FUNCTION_BLOCK Robot_MH

VAR_INPUT
	Robot_1_In			: MH_Robot;
	Part_Unload_Comp	: BOOL;
END_VAR

VAR_OUTPUT
	Robot_1_Out			: MH_Robot;	
END_VAR

VAR
	Pickup_Delay			: ARRAY [0..5] OF TON;
END_VAR

CASE Robot_1_In.i_Prg_No OF
	101:
		IF (Robot_1_In.i_Home AND Robot_1_In.i_Area_Ok1 AND Robot_1_In.i_Start) THEN
		Pickup_Delay[0](IN:= Robot_1_In.i_Start, PT:= T#1S, Q=> , ET=> );
		IF Pickup_Delay[0].Q THEN
		Robot_1_In.i_Home := FALSE;
		Robot_1_Out.o_Pickup_Comp1 := TRUE;
		Robot_1_In.i_Home := TRUE;
		END_IF
		END_IF
		IF (Robot_1_In.i_Home AND Robot_1_In.i_Area_Ok2 AND Robot_1_In.i_Start) THEN
		Pickup_Delay[1](IN:= Robot_1_In.i_Start, PT:= T#1S, Q=> , ET=> );
		IF Pickup_Delay[1].Q THEN
		Robot_1_In.i_Home := FALSE;
		Robot_1_Out.o_Pickup_Comp2 := TRUE;
		Robot_1_In.i_Home := TRUE;
		END_IF
		END_IF
		IF (Robot_1_In.i_Home AND Part_Unload_Comp) THEN
		Robot_1_Out.o_Pickup_Comp1 := FALSE;
		Robot_1_Out.o_Pickup_Comp2 := FALSE;	
		END_IF
	102:
		IF (Robot_1_In.i_Home AND Robot_1_In.i_Area_Ok1 AND Robot_1_In.i_Start) THEN
		Pickup_Delay[2](IN:= Robot_1_In.i_Start, PT:= T#1S, Q=> , ET=> );
		IF Pickup_Delay[2].Q THEN
		Robot_1_In.i_Home := FALSE;
		Robot_1_Out.o_Pickup_Comp1 := TRUE;
		Robot_1_In.i_Home := TRUE;
		END_IF
		END_IF
		IF (Robot_1_In.i_Home AND Robot_1_In.i_Area_Ok2 AND Robot_1_In.i_Start) THEN
		Pickup_Delay[3](IN:= Robot_1_In.i_Start, PT:= T#1S, Q=> , ET=> );
		IF Pickup_Delay[3].Q THEN
		Robot_1_In.i_Home := FALSE;
		Robot_1_Out.o_Pickup_Comp2 := TRUE;
		Robot_1_In.i_Home := TRUE;
		END_IF
		END_IF
		IF (Robot_1_In.i_Home AND Part_Unload_Comp) THEN
		Robot_1_Out.o_Pickup_Comp1 := FALSE;
		Robot_1_Out.o_Pickup_Comp2 := FALSE;	
		END_IF
END_CASE

END_FUNCTION_BLOCK

(* stored: Version 1.1.0.1, ProductVersion 3.1.4024.16
   POU Robot_MH: Id {60b6a47e-c8b3-45c6-bc55-0a26b034c2df}, SpecialFunc None *)
